RoboDK station: Demo_Digital_Twin.rdk

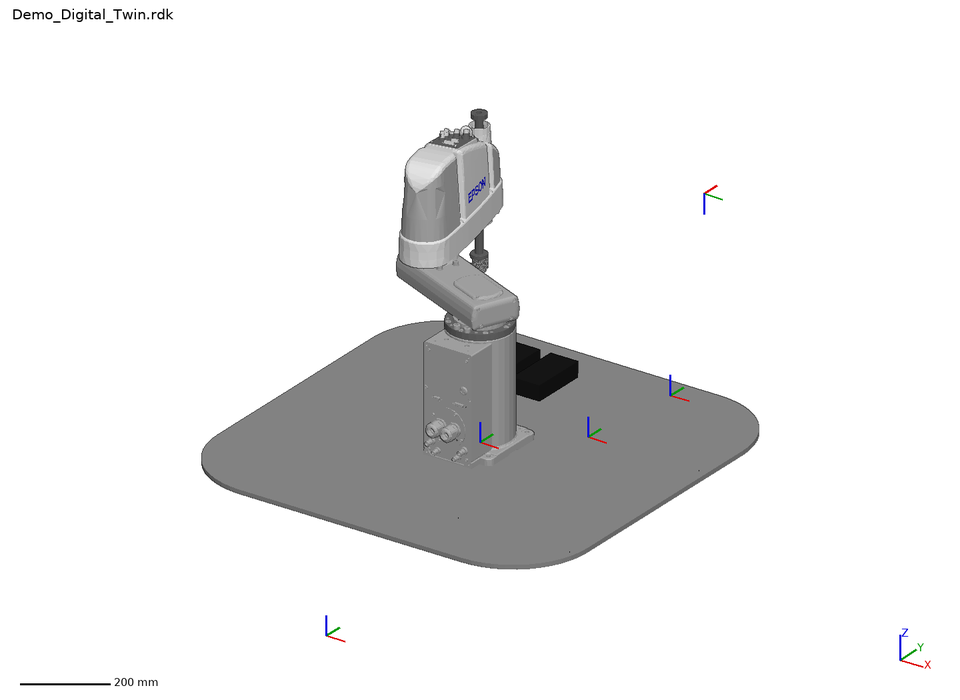
[picture v0: the station drawn from its stored meshes, robots at their saved joint values, targets as dots, program paths as lines]
Station Demo_Digital_Twin (saved by RoboDK 5.9.6). Poses are relative to the parent item; angles as X-Y-Z fixed-axis rotations.
  - frame Epson_G6_451s Base at (0, 0, 0) mm
    - robot Epson_G6_451s: 4 axes
        modified DH rows (alpha deg, a mm, theta deg, d mm): 0, 0, 0, 0; 0, 200, 0, 0; 0, 250, 0, -180 linear; 180, 0, 0, 0
        joint limits [-62, -142, -180, -360] to [242, 142, 0, 360]; home [0, 0, 0, 0]; saved at [156.626, -55.927, -65, -79.301]
      - tool VacuumGripper, TCP at (0, 0, 94) mm, size 51.8 x 37 x 129 mm, geometry from VacuumGripper.step
    - object WorkSurface at (0, 0, 0) mm, size 1000 x 1000 x 10 mm, geometry from WorkSurface.step
  - frame Camera Frame at (560.73, 64.2, 743.82) mm, rotated rx 180 ry 0 rz 90 deg
    - camera Camera 1
  - frame Frame 3 at (281.44, -994.11, 0) mm
    - object TestMovementPiece1 at (0, 0, 0) mm, size 150 x 75 x 40 mm, geometry from TestMovementPiece.step
  - Python program DemoMoveBlocks (listed below)
  - frame Frame 5 at (180, 160, 0) mm
    - object 1 at (0, 0, 0) mm, size 2 x 2 x 2 mm, geometry from Calibration Dots.step
    - object 2 at (0, -500, 0) mm, size 2 x 2 x 2 mm, geometry from Calibration Dots.step
    - object 3 at (300, -500, 0) mm, size 2 x 2 x 2 mm, geometry from Calibration Dots.step
    - object 4 at (300, 0, 0) mm, size 2 x 2 x 2 mm, geometry from Calibration Dots.step
  - frame Frame 6 at (517.85, -4.4, 262.44) mm
  - Python program Prog2 (listed below)
  - Python program DemoWorking (listed below)
  - program Attach (1 instructions, listed below)
  - program Detach (1 instructions, listed below)
  - object TestMovementPiece4 at (-48.37, 319.86, 0) mm, rotated rx 0 ry 0 rz -89.96 deg, size 150 x 75 x 40 mm, geometry from TestMovementPiece.step
  - object TestMovementPiece3 at (-152.85, 320.13, 0) mm, rotated rx 0 ry 0 rz -90.01 deg, size 150 x 75 x 40 mm, geometry from TestMovementPiece.step
  - object TestMovementPiece2 at (-238.82, 314.45, 0) mm, rotated rx 0 ry 0 rz -89.74 deg, size 150 x 75 x 40 mm, geometry from TestMovementPiece.step

--- Python program DemoMoveBlocks ---
from robodk import robolink, robomath
from robodk.robolink import ITEM_TYPE_CAMERA, ITEM_TYPE_ROBOT
import numpy as np
import cv2 as cv

RDK = robolink.Robolink()

# ----------------------------
# User config
# ----------------------------
CAM_NAME = "Camera 1"
WINDOW_NAME = "RoboDK Vision (C=Calibrate, M=Move to BLACK, ESC=Quit)"

ROBOT_NAME = "Epson_G6_451s"
robot = RDK.Item(ROBOT_NAME, ITEM_TYPE_ROBOT)
if not robot.Valid():
    raise Exception(f"Robot not found: {ROBOT_NAME}. Rename ROBOT_NAME to match your RoboDK station tree.")

# If you want to KEEP current orientation, set this False
APPLY_DETECTED_ANGLE = True

# Optional: tool rotation offset (deg) if your tool zero doesn’t match camera angle
TOOL_ANGLE_OFFSET_DEG = 0.0

# ----------------------------
# Camera connect
# ----------------------------
cam_item = RDK.Item(CAM_NAME, ITEM_TYPE_CAMERA)
if not cam_item.Valid():
    raise Exception(f"Camera not found: {CAM_NAME}")

cam_item.setParam("Open", 1)

# ----------------------------
# Homography world points (mm)
# Click in this exact order:
# 1) (180, 160)
# 2) (180, -340)
# 3) (480, -340)
# 4) (480, 160)
# ----------------------------
WORLD_PTS_MM = np.array([
    [180.0,  160.0],
    [180.0, -340.0],
    [480.0, -340.0],
    [480.0,  160.0],
], dtype=np.float32)

# ----------------------------
# Detection tuning
# ----------------------------
MIN_AREA_PX = 800
MAX_AREA_PX = 10_000_000
RECTANGULARITY_MIN = 0.70

PRINT_EVERY_N_FRAMES = 10
frame_idx = 0

# ----------------------------
# Calibration state
# ----------------------------
H = None
calib_mode = False
clicked_pts = []
freeze_img = None

def snapshot_bgr():
    bytes_img = RDK.Cam2D_Snapshot("", cam_item)
    if not isinstance(bytes_img, bytes) or bytes_img == b"":
        return None
    nparr = np.frombuffer(bytes_img, np.uint8)
    return cv.imdecode(nparr, cv.IMREAD_COLOR)

def rect_angle_degrees(rect):
    (cx, cy), (w, h), ang = rect
    if w < h:
        ang += 90.0
    return ang

def pixel_to_world(cx, cy, Hmat):
    pt = np.array([[[cx, cy]]], dtype=np.float32)
    XY = cv.perspectiveTransform(pt, Hmat)[0][0]
    return float(XY[0]), float(XY[1])

def find_rectangles_from_mask(mask):
    kernel = np.ones((7, 7), np.uint8)
    mask = cv.morphologyEx(mask, cv.MORPH_OPEN, kernel, iterations=2)
    mask = cv.morphologyEx(mask, cv.MORPH_CLOSE, kernel, iterations=3)

    contours, _ = cv.findContours(mask, cv.RETR_EXTERNAL, cv.CHAIN_APPROX_SIMPLE)

    rects = []
    for cnt in contours:
        area = cv.contourArea(cnt)
        if area < MIN_AREA_PX or area > MAX_AREA_PX:
            continue

        rect = cv.minAreaRect(cnt)
        (cx, cy), (w, h), _ = rect
        if w <= 2 or h <= 2:
            continue

        rect_area = w * h
        rectangularity = area / (rect_area + 1e-6)
        if rectangularity < RECTANGULARITY_MIN:
            continue

        rects.append(rect)

    return rects

def build_color_masks(img_bgr):
    hsv = cv.cvtColor(img_bgr, cv.COLOR_BGR2HSV)

    black_lower = np.array([0, 0, 0], dtype=np.uint8)
    black_upper = np.array([180, 255, 60], dtype=np.uint8)
    mask_black = cv.inRange(hsv, black_lower, black_upper)

    red1_lower = np.array([0, 40, 30], dtype=np.uint8)
    red1_upper = np.array([15, 255, 255], dtype=np.uint8)
    red2_lower = np.array([165, 40, 30], dtype=np.uint8)
    red2_upper = np.array([180, 255, 255], dtype=np.uint8)
    mask_red = cv.inRange(hsv, red1_lower, red1_upper) | cv.inRange(hsv, red2_lower, red2_upper)

    return mask_black, mask_red

def draw_calib_overlay(img):
    out = img.copy()
    cv.putText(out, "CALIB MODE: click 4 points (1..4) in order. ESC=Quit",
               (10, 30), cv.FONT_HERSHEY_SIMPLEX, 0.8, (0, 255, 255), 2)

    y0 = 60
    for i, p in enumerate(WORLD_PTS_MM, start=1):
        cv.putText(out, f"{i}: world({p[0]:.0f},{p[1]:.0f})",
                   (10, y0 + 25*(i-1)), cv.FONT_HERSHEY_SIMPLEX, 0.7, (0, 255, 255), 2)

    for i, (x, y) in enumerate(clicked_pts, start=1):
        cv.circle(out, (int(x), int(y)), 6, (0, 255, 255), -1)
        cv.putText(out, str(i), (int(x) + 10, int(y) - 10),
                   cv.FONT_HERSHEY_SIMPLEX, 0.9, (0, 255, 255), 2)

    return out

def on_mouse(event, x, y, flags, param):
    global clicked_pts, H, calib_mode, freeze_img

    if event != cv.EVENT_LBUTTONDOWN:
        return
    if not calib_mode or freeze_img is None:
        return

    clicked_pts.append([x, y])
    print(f"Clicked {len(clicked_pts)}/4: ({x},{y})")

    if len(clicked_pts) == 4:
        pix = np.array(clicked_pts, dtype=np.float32)
        H_new, _ = cv.findHomography(pix, WORLD_PTS_MM)

        if H_new is None:
            print("Homography failed. Press C and try again.")
            H = None
        else:
            H = H_new
            print("Homography computed (pixel -> world mm):")
            print(H)

        calib_mode = False
        freeze_img = None
        clicked_pts = []

def move_to_black(best_black_rect):
    if H is None:
        print("Not calibrated. Press C first.")
        return
    if best_black_rect is None:
        print("No black rectangle detected.")
        return

    (cx, cy), (_, _), _ = best_black_rect
    ang_deg = rect_angle_degrees(best_black_rect)
    X_mm, Y_mm = pixel_to_world(cx, cy, H)

    # ---- THIS IS THE IMPORTANT PART: "GO XY" style move ----
    pose_now = robot.Pose()
    xyzrpw = robomath.Pose_2_TxyzRxyz(pose_now)  # [x,y,z,rx,ry,rz] (mm, radians)

    # Replace only X and Y
    xyzrpw[0] = X_mm
    xyzrpw[1] = Y_mm

    # Optionally apply detected angle as a delta about Z (keeps Rx/Ry and Z the same)
    if APPLY_DETECTED_ANGLE:
        xyzrpw[5] = xyzrpw[5] + (ang_deg + TOOL_ANGLE_OFFSET_DEG) * (np.pi / 180.0)

    pose_xy = robomath.TxyzRxyz_2_Pose(xyzrpw)

    print(f"Moving to BLACK (Go-XY style): X={X_mm:.2f} Y={Y_mm:.2f} ang={ang_deg:.2f}")
    robot.MoveJ(pose_xy)

# Create OpenCV window + mouse callback
cv.namedWindow(WINDOW_NAME, cv.WINDOW_NORMAL)
cv.setMouseCallback(WINDOW_NAME, on_mouse)

print("Controls: C=Calibrate, M=Move to BLACK, ESC=Quit")
print("Calibration click order (world points mm):")
for i, p in enumerate(WORLD_PTS_MM, start=1):
    print(f"  {i}: ({p[0]}, {p[1]})")

last_best_black = None

while True:
    # Calibration mode
    if calib_mode and freeze_img is not None:
        calib_view = draw_calib_overlay(freeze_img)
        cv.imshow(WINDOW_NAME, calib_view)
        key = cv.waitKey(20) & 0xFF
        if key == 27:
            break
        continue

    img = snapshot_bgr()
    if img is None:
        break

    frame_idx += 1
    do_print = (frame_idx % PRINT_EVERY_N_FRAMES == 0)

    mask_black, mask_red = build_color_masks(img)
    rects_black = find_rectangles_from_mask(mask_black)
    rects_red = find_rectangles_from_mask(mask_red)

    last_best_black = max(rects_black, key=lambda r: r[1][0] * r[1][1]) if rects_black else None

    detections = [("BLACK", r) for r in rects_black] + [("RED", r) for r in rects_red]
    detections.sort(key=lambda d: d[1][1][0] * d[1][1][1], reverse=True)

    if H is None:
        cv.putText(img, "NOT CALIBRATED: Press C", (10, 30),
                   cv.FONT_HERSHEY_SIMPLEX, 0.9, (0, 255, 255), 2)
    else:
        cv.putText(img, "Calibrated. Press M to move to BLACK", (10, 30),
                   cv.FONT_HERSHEY_SIMPLEX, 0.9, (0, 255, 255), 2)

    if do_print and detections:
        print("---- Frame detections ----")

    for i, (label, rect) in enumerate(detections):
        (cx, cy), (w, h), _ = rect
        ang = rect_angle_degrees(rect)

        box = cv.boxPoints(rect).astype(np.int32)
        cv.drawContours(img, [box], 0, (0, 255, 0), 2)
        cv.circle(img, (int(cx), int(cy)), 4, (255, 255, 255), -1)

        if H is not None:
            X_mm, Y_mm = pixel_to_world(cx, cy, H)
            text = f"{label} X={X_mm:.1f} Y={Y_mm:.1f} A={ang:.1f}"
            if do_print:
                print(f"{label} {i}: X={X_mm:.2f} Y={Y_mm:.2f} A={ang:.2f}")
        else:
            text = f"{label} px=({cx:.0f},{cy:.0f}) A={ang:.1f}"

        if label == "BLACK" and rect is last_best_black:
            cv.putText(img, "TARGET", (int(cx) - 30, int(cy) + 30),
                       cv.FONT_HERSHEY_SIMPLEX, 0.8, (0, 255, 255), 2)

        cv.putText(img, text, (int(cx) + 10, int(cy) - 10),
                   cv.FONT_HERSHEY_SIMPLEX, 0.6, (0, 255, 0), 2)

    cv.imshow(WINDOW_NAME, img)

    key = cv.waitKey(1) & 0xFF
    if key == 27:
        break
    if key in (ord('c'), ord('C')):
        calib_mode = True
        freeze_img = img.copy()
        clicked_pts = []
        print("Calibration mode: click 4 points now...")
    if key in (ord('m'), ord('M')):
        move_to_black(last_best_black)

    if cv.getWindowProperty(WINDOW_NAME, cv.WND_PROP_VISIBLE) < 1:
        break

cv.destroyAllWindows()
RDK.Cam2D_Close(cam_item)

--- Python program Prog2 ---
from robodk import robolink, robomath
from robodk.robolink import ITEM_TYPE_ROBOT

RDK = robolink.Robolink()

ROBOT_NAME = "Epson_G6_451s"  # change to your robot name in RoboDK station tree
robot = RDK.Item(ROBOT_NAME, ITEM_TYPE_ROBOT)
if not robot.Valid():
    raise Exception(f"Robot not found: {ROBOT_NAME}")

# Desired XY (mm)
X = 287.600
Y = -4.400

# Get current robot pose (keeps current Z + orientation)
pose = robot.Pose()
xyzrpw = robomath.Pose_2_TxyzRxyz(pose)  # [x,y,z,rx,ry,rz] in mm and radians

# Replace only X and Y
xyzrpw[0] = X
xyzrpw[1] = Y

pose_xy = robomath.TxyzRxyz_2_Pose(xyzrpw)

RDK.ShowMessage(f"Moving to XY: ({X:.3f}, {Y:.3f}) keeping Z={xyzrpw[2]:.3f}", False)

# Move (use MoveJ to be more forgiving)
robot.MoveJ(pose_xy)

RDK.ShowMessage("Done.", False)

--- Python program DemoWorking ---
from robodk import robolink, robomath
from robodk.robolink import ITEM_TYPE_CAMERA, ITEM_TYPE_ROBOT, ITEM_TYPE_TOOL, TargetReachError
import numpy as np
import cv2 as cv
import time

RDK = robolink.Robolink()

# ============================================================
# USER CONFIG
# ============================================================
CAM_NAME = "Camera 1"
ROBOT_NAME = "Epson_G6_451s"
TOOL_NAME = "VacuumGripper"

WINDOW_NAME = "RoboDK Vision (C=Calibrate, M=Pick/Place Selected, P=Auto, ESC=Quit)"
MASK_WINDOW = "Mask"
CONTROL_WINDOW = "Controls"

robot = RDK.Item(ROBOT_NAME, ITEM_TYPE_ROBOT)
if not robot.Valid():
    raise Exception(f"Robot not found: {ROBOT_NAME}")

cam_item = RDK.Item(CAM_NAME, ITEM_TYPE_CAMERA)
if not cam_item.Valid():
    raise Exception(f"Camera not found: {CAM_NAME}")

named_tool = RDK.Item(TOOL_NAME)
if not named_tool.Valid():
    raise Exception(f"[ERROR] Tool '{TOOL_NAME}' not found in the RoboDK station.")

print(f"[INFO] Using named tool: {named_tool.Name()}")

# Set the robot TCP using the named tool
robot.setPoseTool(named_tool)

# Get the active tool link actually associated with the robot
tool = robot.getLink(ITEM_TYPE_TOOL)
if not tool.Valid():
    raise Exception("[ERROR] Robot active tool link is not valid after setPoseTool().")

print(f"[INFO] Active robot tool link: {tool.Name()}")

cam_item.setParam("Open", 1)

# ============================================================
# CALIBRATION WORLD POINTS
# These are already relative to the robot base frame
# Click image points in this exact order
# ============================================================
AUTO_WORLD_PTS = np.array([
    [180.0,  160.0],
    [180.0, -340.0],
    [480.0, -340.0],
    [480.0,  160.0],
], dtype=np.float32)

WORLD_W = 1200.0
WORLD_H = 900.0
FLIP_Y = False

# Optional offsets after homography mapping
ROBOT_X_OFFSET = 0.0
ROBOT_Y_OFFSET = 0.0
ROBOT_U_OFFSET = 0.0

# ============================================================
# ROBOT MOTION SETTINGS
# ============================================================
HOME_JOINTS = [90.0, 0.0, 0.0, 0.0]

PICK_Z_ABOVE = 141.0
PICK_Z_DOWN = 37.0

DROP_U = 180.0
DROP_Z_ABOVE = 141.0
DROP_Z_DOWN = 37.0

DROP_POINTS = [
    (-60.0, 325.0),
    (-145.0, 325.0),
    (-230.0, 325.0),
]

WAIT_AT_DROP_S = 0.5
APPLY_DETECTED_ANGLE = True

# ============================================================
# DETECTION SETTINGS
# ============================================================
PROC_WIDTH = 1280

DARK_THRESHOLD = 21
BLUR_K = 5
MORPH_K = 0
MORPH_ITERS = 2
MIN_AREA_FRAC = 0.0003
MAX_AREA_FRAC = 0.10
MIN_FILL_RATIO = 0.45

SEND_PERIOD = 0.5
MIN_MOVE_MM = 5.0
AUTO_RUN = False

# ============================================================
# GLOBAL STATE
# ============================================================
H = None
calib_mode = False
clicked_pts = []
freeze_img = None

frame_idx = 0
movecount = 0
last_cmd = None
last_xy = None
last_sent_t = 0.0
busy = False

# ============================================================
# CAMERA
# ============================================================
def snapshot_bgr():
    bytes_img = RDK.Cam2D_Snapshot("", cam_item)
    if not isinstance(bytes_img, bytes) or bytes_img == b"":
        return None
    nparr = np.frombuffer(bytes_img, np.uint8)
    return cv.imdecode(nparr, cv.IMREAD_COLOR)

# ============================================================
# TOOL HELPERS
# ============================================================
def refresh_active_tool():
    """Refresh the active tool link from the robot."""
    global tool
    tool = robot.getLink(ITEM_TYPE_TOOL)
    if not tool.Valid():
        print("[ERROR] Active robot tool link is not valid.")
        return False
    return True


# ============================================================
# VACUUM / ATTACH-DETACH
# ============================================================
def vacuum_on():
    """
    Attach the closest object to the ACTIVE tool,
    same approach as RoboDK example TCP_On().
    """
    try:
        if not refresh_active_tool():
            return False

        tool.AttachClosest()
        RDK.RunMessage("Vacuum ON")
        print(f"[VAC] ON using tool: {tool.Name()}")
        return True

    except Exception as e:
        print(f"[ERROR] Vacuum ON failed: {e}")
        return False


def vacuum_off(itemleave=0):
    """
    Detach objects from the ACTIVE tool,
    same approach as RoboDK example TCP_Off().
    """
    try:
        if not refresh_active_tool():
            return False

        tool.DetachAll(itemleave)
        RDK.RunMessage("Vacuum OFF")
        print(f"[VAC] OFF using tool: {tool.Name()}")
        return True

    except Exception as e:
        print(f"[ERROR] Vacuum OFF failed: {e}")
        return False

# ============================================================
# UI CONTROLS
# ============================================================
def setup_tuning_sliders(window_name: str):
    cv.namedWindow(window_name, cv.WINDOW_NORMAL)
    cv.resizeWindow(window_name, 420, 300)

    cv.createTrackbar("Dark threshold", window_name, DARK_THRESHOLD, 255, lambda v: None)
    cv.createTrackbar("Blur k (odd)", window_name, BLUR_K, 31, lambda v: None)
    cv.createTrackbar("Max area x1e6", window_name, int(MAX_AREA_FRAC * 1_000_000), 1000000, lambda v: None)
    cv.createTrackbar("Morph k (odd)", window_name, MORPH_K, 51, lambda v: None)
    cv.createTrackbar("Morph iters", window_name, MORPH_ITERS, 10, lambda v: None)
    cv.createTrackbar("Min area x1e6", window_name, int(MIN_AREA_FRAC * 1_000_000), 200000, lambda v: None)
    cv.createTrackbar("Min fill x100", window_name, int(MIN_FILL_RATIO * 100), 100, lambda v: None)

def read_tuning_sliders(window_name: str):
    global DARK_THRESHOLD, BLUR_K, MORPH_K, MORPH_ITERS, MIN_AREA_FRAC, MAX_AREA_FRAC, MIN_FILL_RATIO

    DARK_THRESHOLD = cv.getTrackbarPos("Dark threshold", window_name)

    BLUR_K = cv.getTrackbarPos("Blur k (odd)", window_name)
    if BLUR_K < 1:
        BLUR_K = 1
    if BLUR_K % 2 == 0:
        BLUR_K += 1

    MORPH_K = cv.getTrackbarPos("Morph k (odd)", window_name)
    if MORPH_K < 0:
        MORPH_K = 0
    if MORPH_K > 0 and MORPH_K % 2 == 0:
        MORPH_K += 1

    MORPH_ITERS = cv.getTrackbarPos("Morph iters", window_name)
    MIN_AREA_FRAC = cv.getTrackbarPos("Min area x1e6", window_name) / 1_000_000.0
    MAX_AREA_FRAC = cv.getTrackbarPos("Max area x1e6", window_name) / 1_000_000.0
    MIN_FILL_RATIO = cv.getTrackbarPos("Min fill x100", window_name) / 100.0

# ============================================================
# CALIBRATION
# ============================================================
def draw_calib_overlay(img):
    out = img.copy()
    cv.putText(
        out,
        "CALIB MODE: click 4 points in order, C computes, R resets, ESC quits",
        (10, 30),
        cv.FONT_HERSHEY_SIMPLEX,
        0.7,
        (0, 255, 255),
        2,
    )

    y0 = 60
    for i, p in enumerate(AUTO_WORLD_PTS, start=1):
        cv.putText(
            out,
            f"{i}: world({p[0]:.1f}, {p[1]:.1f})",
            (10, y0 + 25 * (i - 1)),
            cv.FONT_HERSHEY_SIMPLEX,
            0.6,
            (0, 255, 255),
            2,
        )

    for i, (x, y) in enumerate(clicked_pts, start=1):
        cv.circle(out, (int(x), int(y)), 6, (0, 255, 255), -1)
        cv.putText(
            out,
            str(i),
            (int(x) + 10, int(y) - 10),
            cv.FONT_HERSHEY_SIMPLEX,
            0.8,
            (0, 255, 255),
            2,
        )

    return out

def on_mouse(event, x, y, flags, param):
    global clicked_pts
    if event == cv.EVENT_LBUTTONDOWN and calib_mode and freeze_img is not None:
        if len(clicked_pts) < 4:
            clicked_pts.append([float(x), float(y)])
            print(f"Clicked point {len(clicked_pts)}: ({x}, {y})")

def compute_homography():
    global H, calib_mode, freeze_img, clicked_pts

    if len(clicked_pts) != 4:
        print("Need exactly 4 clicked points.")
        return

    pix = np.array(clicked_pts, dtype=np.float32)
    H_new, _ = cv.findHomography(pix, AUTO_WORLD_PTS)

    if H_new is None:
        print("Homography failed.")
        H = None
    else:
        H = H_new.astype(np.float32)
        print("Homography computed.")
        print(H)

    calib_mode = False
    freeze_img = None
    clicked_pts = []

# ============================================================
# DETECTION
# ============================================================
def rect_angle_to_u(angle_deg: float, rw: float, rh: float) -> float:
    u = float(angle_deg)
    if rw < rh:
        u = u + 90.0
    if u < 0:
        u += 180.0
    return float(u)

def detect_rectangles(frame_bgr, homography):
    h_full, w_full = frame_bgr.shape[:2]

    proc_w = PROC_WIDTH
    proc_h = int((proc_w * h_full) / w_full)
    proc = cv.resize(frame_bgr, (proc_w, proc_h))

    gray = cv.cvtColor(proc, cv.COLOR_BGR2GRAY)
    gray = cv.GaussianBlur(gray, (int(BLUR_K), int(BLUR_K)), 0)

    _, mask = cv.threshold(gray, int(DARK_THRESHOLD), 255, cv.THRESH_BINARY_INV)

    if MORPH_K > 1 and MORPH_ITERS > 0:
        kernel = cv.getStructuringElement(cv.MORPH_RECT, (int(MORPH_K), int(MORPH_K)))
        mask = cv.morphologyEx(mask, cv.MORPH_CLOSE, kernel, iterations=int(MORPH_ITERS))

    contours, _ = cv.findContours(mask, cv.RETR_EXTERNAL, cv.CHAIN_APPROX_SIMPLE)

    proc_area = float(proc_w * proc_h)
    area_min = max(400.0, float(MIN_AREA_FRAC) * proc_area)
    area_max = float(MAX_AREA_FRAC) * proc_area

    scale_x = w_full / proc_w
    scale_y = h_full / proc_h

    detections = []

    for cnt in contours:
        area = cv.contourArea(cnt)
        if area < area_min or area > area_max:
            continue

        rect = cv.minAreaRect(cnt)
        (_, _), (rw, rh), raw_angle = rect

        if rw <= 1 or rh <= 1:
            continue

        rect_area = float(rw * rh)
        if rect_area <= 1:
            continue

        fill_ratio = float(area) / rect_area
        if fill_ratio < float(MIN_FILL_RATIO):
            continue

        box_proc = cv.boxPoints(rect).astype(np.float32)
        box_full = np.array([[pt[0] * scale_x, pt[1] * scale_y] for pt in box_proc], dtype=np.int32)

        (cxp, cyp), _, _ = rect
        cx = cxp * scale_x
        cy = cyp * scale_y

        if homography is None:
            continue

        center_pixel = np.array([[[cx, cy]]], dtype=np.float32)
        real_pt = cv.perspectiveTransform(center_pixel, homography)
        rx, ry = real_pt[0][0]

        if FLIP_Y:
            ry = WORLD_H - ry

        u_deg = rect_angle_to_u(raw_angle, rw, rh)
        score = area * fill_ratio

        detections.append({
            "score": float(score),
            "area": float(area),
            "fill_ratio": float(fill_ratio),
            "box": box_full,
            "center_px": (float(cx), float(cy)),
            "center_mm": (float(rx), float(ry)),
            "u_deg": float(u_deg),
            "rect_wh": (float(rw), float(rh)),
        })

    detections.sort(key=lambda d: (-d["score"], -d["area"], d["center_px"][0], d["center_px"][1]))

    return {
        "mask": mask,
        "detections": detections
    }

# ============================================================
# ROBOT POSE HELPERS
# ============================================================
def pose_with_xyzu(x_mm, y_mm, z_mm, u_deg):
    pose_now = robot.Pose()
    xyzrpw = list(robomath.Pose_2_TxyzRxyz(pose_now))

    xyzrpw[0] = float(x_mm)
    xyzrpw[1] = float(y_mm)
    xyzrpw[2] = float(z_mm)

    if APPLY_DETECTED_ANGLE:
        xyzrpw[5] = np.deg2rad(float(u_deg))

    pose_new = robomath.TxyzRxyz_2_Pose(xyzrpw)
    return pose_new

def explain_move_error(err, x_mm, y_mm, z_mm, u_deg, linear):
    move_type = "MoveL" if linear else "MoveJ"
    print(f"[ERROR] {move_type} failed.")
    print(f"[ERROR] Requested pose: X={x_mm:.2f} Y={y_mm:.2f} Z={z_mm:.2f} U={u_deg:.2f}")

    try:
        pose_now = robot.Pose()
        xyzrpw_now = list(robomath.Pose_2_TxyzRxyz(pose_now))
        print(
            f"[ERROR] Current pose: "
            f"X={xyzrpw_now[0]:.2f} Y={xyzrpw_now[1]:.2f} Z={xyzrpw_now[2]:.2f} "
            f"RZ={np.rad2deg(xyzrpw_now[5]):.2f} deg"
        )
    except Exception:
        print("[ERROR] Could not read current robot pose.")

    print(f"[ERROR] RoboDK message: {err}")

    if linear:
        print("[ERROR] Likely issue: the straight-line path is not reachable from the current robot position.")
    else:
        print("[ERROR] Likely issue: RoboDK could not find a valid joint solution for that target pose.")

def move_xyzu(x_mm, y_mm, z_mm, u_deg, linear=False):
    pose = pose_with_xyzu(x_mm, y_mm, z_mm, u_deg)

    try:
        if linear:
            robot.MoveL(pose)
        else:
            robot.MoveJ(pose)
        return True

    except TargetReachError as e:
        explain_move_error(e, x_mm, y_mm, z_mm, u_deg, linear)
        return False

    except Exception as e:
        print("[ERROR] Unexpected robot move failure.")
        explain_move_error(e, x_mm, y_mm, z_mm, u_deg, linear)
        return False


# ============================================================
# PICK / PLACE LOGIC
# ============================================================
def run_pick_place(x_cmd, y_cmd, u_cmd):
    global movecount, busy

    if busy:
        return False

    busy = True
    try:
        print(f"[PICK] Target X={x_cmd:.2f} Y={y_cmd:.2f} U={u_cmd:.2f}")

        # Move above pick point
        if not move_xyzu(x_cmd, y_cmd, PICK_Z_ABOVE, u_cmd, linear=False):
            print("[ABORT] Could not move above pick point.")
            return False

        # Move down to pick point
        if not move_xyzu(x_cmd, y_cmd, PICK_Z_DOWN, u_cmd, linear=True):
            print("[ABORT] Could not move down to pick point.")
            return False

        # Attach object
        if not vacuum_on():
            print("[ABORT] Could not attach block.")
            return False

        time.sleep(WAIT_AT_DROP_S)

        # Lift object
        if not move_xyzu(x_cmd, y_cmd, PICK_Z_ABOVE, u_cmd, linear=True):
            print("[ABORT] Could not lift object after pick.")
            return False

        # Determine drop point
        movecount += 1
        if movecount == 1:
            dx, dy = DROP_POINTS[0]
        elif movecount == 2:
            dx, dy = DROP_POINTS[1]
        elif movecount == 3:
            dx, dy = DROP_POINTS[2]
        else:
            movecount = 1
            dx, dy = DROP_POINTS[0]

        print(f"[PLACE] movecount={movecount} -> drop X={dx:.2f} Y={dy:.2f} U={DROP_U:.2f}")

        # Move above drop point
        if not move_xyzu(dx, dy, DROP_Z_ABOVE, DROP_U, linear=False):
            print("[ABORT] Could not move above drop point.")
            return False

        # Move down to drop point
        if not move_xyzu(dx, dy, DROP_Z_DOWN, DROP_U, linear=True):
            print("[ABORT] Could not move down to drop point.")
            return False

        # Detach object
        if not vacuum_off():
            print("[ABORT] Could not detach block.")
            return False

        time.sleep(WAIT_AT_DROP_S)

        # Lift after drop
        if not move_xyzu(dx, dy, DROP_Z_ABOVE, DROP_U, linear=True):
            print("[ABORT] Could not lift after drop.")
            return False

        print("[DONE] Pick/place completed successfully.")
        return True

    finally:
        busy = False

# ============================================================
# MAIN
# ============================================================
cv.namedWindow(WINDOW_NAME, cv.WINDOW_NORMAL)
cv.namedWindow(MASK_WINDOW, cv.WINDOW_NORMAL)
cv.setMouseCallback(WINDOW_NAME, on_mouse)
setup_tuning_sliders(CONTROL_WINDOW)

print("Controls:")
print("  C = start calibration from frozen frame")
print("  M = pick/place selected block once")
print("  P = toggle auto pick/place")
print("  H = home robot")
print("  R = reset movecount to 0")
print("  ESC = quit")

try:
    robot.MoveJ(HOME_JOINTS)
except Exception as e:
    print(f"[WARN] Home move failed: {e}")

while True:
    if calib_mode and freeze_img is not None:
        calib_view = draw_calib_overlay(freeze_img)
        cv.imshow(WINDOW_NAME, calib_view)
        key = cv.waitKey(20) & 0xFF

        if key == 27:
            break
        elif key in (ord('r'), ord('R')):
            clicked_pts = []
            print("Calibration points reset.")
        elif key in (ord('c'), ord('C')):
            compute_homography()

        continue

    img = snapshot_bgr()
    if img is None:
        print("Camera snapshot failed.")
        break

    read_tuning_sliders(CONTROL_WINDOW)
    result = detect_rectangles(img, H)

    cv.imshow(MASK_WINDOW, result.get("mask", np.zeros((10, 10), dtype=np.uint8)))

    disp = img.copy()
    detections = result.get("detections", [])

    status = "AUTO: ON" if AUTO_RUN else "AUTO: OFF"
    color = (0, 255, 0) if AUTO_RUN else (0, 0, 255)
    cv.putText(disp, status, (20, 35), cv.FONT_HERSHEY_SIMPLEX, 1.0, color, 3)

    cv.putText(
        disp,
        f"movecount={movecount}",
        (20, 70),
        cv.FONT_HERSHEY_SIMPLEX,
        0.8,
        (255, 255, 255),
        2
    )

    cv.putText(
        disp,
        f"thr={DARK_THRESHOLD} blur={BLUR_K} morph={MORPH_K} iters={MORPH_ITERS}",
        (20, 100),
        cv.FONT_HERSHEY_SIMPLEX,
        0.6,
        (255, 255, 255),
        2
    )

    cv.putText(
        disp,
        f"minArea={MIN_AREA_FRAC:.6f} maxArea={MAX_AREA_FRAC:.6f} minFill={MIN_FILL_RATIO:.2f}",
        (20, 125),
        cv.FONT_HERSHEY_SIMPLEX,
        0.6,
        (255, 255, 255),
        2
    )

    if H is None:
        cv.putText(
            disp,
            "NOT CALIBRATED - press C",
            (20, 155),
            cv.FONT_HERSHEY_SIMPLEX,
            0.8,
            (0, 255, 255),
            2
        )
    else:
        cv.putText(
            disp,
            "Calibrated",
            (20, 155),
            cv.FONT_HERSHEY_SIMPLEX,
            0.8,
            (0, 255, 0),
            2
        )

    selected_cmd = None

    if detections:
        cv.putText(
            disp,
            f"Detected boxes: {len(detections)}",
            (20, 185),
            cv.FONT_HERSHEY_SIMPLEX,
            0.8,
            (0, 255, 255),
            2
        )

        for i, det in enumerate(detections):
            box = det["box"]
            cx, cy = det["center_px"]
            rx, ry = det["center_mm"]
            u_deg = det["u_deg"]

            is_selected = (i == 0)
            box_color = (0, 255, 0) if is_selected else (255, 200, 0)
            center_color = (0, 0, 255) if is_selected else (255, 0, 0)
            thickness = 4 if is_selected else 2

            cv.drawContours(disp, [box], 0, box_color, thickness)
            cv.circle(disp, (int(cx), int(cy)), 6, center_color, -1)

            label = f"#{i+1} X={rx:.1f} Y={ry:.1f} U={u_deg:.1f}"
            cv.putText(
                disp,
                label,
                (int(cx) - 140, int(cy) - 10),
                cv.FONT_HERSHEY_SIMPLEX,
                0.6,
                box_color,
                2
            )

        target = detections[0]
        rx, ry = target["center_mm"]
        u_deg = target["u_deg"]

        x_cmd = rx + ROBOT_X_OFFSET
        y_cmd = ry + ROBOT_Y_OFFSET
        u_cmd = u_deg + ROBOT_U_OFFSET

        selected_cmd = (x_cmd, y_cmd, u_cmd)
        last_cmd = selected_cmd

        cv.putText(
            disp,
            f"SELECTED -> X={x_cmd:.1f} Y={y_cmd:.1f} U={u_cmd:.1f}",
            (20, 215),
            cv.FONT_HERSHEY_SIMPLEX,
            0.8,
            (0, 255, 0),
            2
        )

        now = time.time()
        moved_enough = True

        if last_xy is not None:
            dx = x_cmd - last_xy[0]
            dy = y_cmd - last_xy[1]
            moved_enough = (dx * dx + dy * dy) ** 0.5 >= MIN_MOVE_MM

        if AUTO_RUN and H is not None and (now - last_sent_t) >= SEND_PERIOD and moved_enough and not busy:
            ok = run_pick_place(x_cmd, y_cmd, u_cmd)
            if ok:
                last_sent_t = now
                last_xy = (x_cmd, y_cmd)

    else:
        cv.putText(
            disp,
            "No target detected",
            (20, 185),
            cv.FONT_HERSHEY_SIMPLEX,
            0.9,
            (0, 0, 255),
            2
        )

    cv.imshow(WINDOW_NAME, disp)

    key = cv.waitKey(1) & 0xFF
    if key == 27:
        break

    elif key in (ord('c'), ord('C')):
        calib_mode = True
        freeze_img = img.copy()
        clicked_pts = []
        print("Calibration mode: click 4 points on the frozen image, then press C again.")

    elif key in (ord('m'), ord('M')):
        if H is None:
            print("Not calibrated. Press C first.")
        elif last_cmd is None:
            print("No target detected.")
        else:
            x_cmd, y_cmd, u_cmd = last_cmd
            ok = run_pick_place(x_cmd, y_cmd, u_cmd)
            if ok:
                last_xy = (x_cmd, y_cmd)
                last_sent_t = time.time()

    elif key in (ord('p'), ord('P')):
        AUTO_RUN = not AUTO_RUN
        print(f"AUTO_RUN = {AUTO_RUN}")

    elif key in (ord('h'), ord('H')):
        print("Moving home.")
        try:
            robot.MoveJ(HOME_JOINTS)
        except Exception as e:
            print(f"[ERROR] Home move failed: {e}")

    elif key in (ord('r'), ord('R')):
        movecount = 0
        print("movecount reset to 0.")

    if cv.getWindowProperty(WINDOW_NAME, cv.WND_PROP_VISIBLE) < 1:
        break

cv.destroyAllWindows()
RDK.Cam2D_Close(cam_item)

--- program Attach (robot Epson_G6_451s) ---
  Attach to VacuumGripper

--- program Detach (robot Epson_G6_451s) ---
  Detach from VacuumGripper
